Staubli VAL3: copyArray.pgx

program copyArray(num& x_nDestArray[] (dimensions=1), num& x_nIndex (dimensions=1), num& x_nSourceArray[] (dimensions=1))
  local num i
begin
  // copies whole x_nSourceArray to the greater or equal x_nDestArray
  // starting from x_nIndex, changes the x_nIndex to point to the
  // position one after the copied elements
  for i=0 to size(x_nSourceArray)-1
    x_nDestArray[x_nIndex+i]=x_nSourceArray[i]
  endFor
  x_nIndex=x_nIndex+size(x_nSourceArray)
end
